// TwinCAT 3 PLC project PLC1
// ProgramVersion: 3.1.4026.24
// libraries:
//   Tc2_MC2, * (Beckhoff Automation GmbH)
//   Tc2_Standard, * (Beckhoff Automation GmbH)
//   Tc2_System, * (Beckhoff Automation GmbH)
//   Tc3_Mc3PlanarMotion, * (Beckhoff Automation GmbH)
//   Tc3_Physics, * (Beckhoff Automation GmbH)
//   Tc3_XPlanarUtility, * (Beckhoff Automation GmbH)
//   XPlanarApplication, * (Beckhoff Automation LLC)
// project tree:
//   GVLs/ GVL.TcGVL (not stored)
//   / PlcTask.TcTTO (not stored)
//   POUs/ MAIN.TcPOU
//   POUs/Utilities/ ErrorStep.TcPOU (not stored), NextMinorStep.TcPOU (not stored), NextStep.TcPOU (not stored)
//   POUs/XPlanarModule/ FB_XPlanarModule.TcPOU
// real-time tasks:
//   TASK XPlanar Task_3: cycle T#250us, priority 1, ADS port 350
//   TASK Job Task: cycle default, priority 2
//   TASK MC-Task (MET): cycle T#2ms, priority 3, ADS port 351
//   TASK MC-Task (MPT): cycle T#10ms, priority 4, ADS port 352
//   TASK PlcTask: cycle T#10ms, priority 20, ADS port 353
// variable links:
//   PLC1/PLC1 Instance <-> XPlanar MC Project/Axes/Mover4220_1
//     PlcTask Inputs/MAIN.XPlanarTable.Movers[1]._Mover.MCTOPLC/ACT <-> McToPlc/ACT
//     PlcTask Inputs/MAIN.XPlanarTable.Movers[1]._Mover.MCTOPLC/COORDMODE <-> McToPlc/COORDMODE
//     PlcTask Inputs/MAIN.XPlanarTable.Movers[1]._Mover.MCTOPLC/SET <-> McToPlc/SET
//     PlcTask Inputs/MAIN.XPlanarTable.Movers[1]._Mover.MCTOPLC/SETONTRACK <-> McToPlc/SETONTRACK
//     PlcTask Inputs/MAIN.XPlanarTable.Movers[1]._Mover.MCTOPLC/STD <-> McToPlc/STD
//     PlcTask Outputs/MAIN.XPlanarTable.Movers[1]._Mover.PLCTOMC/STD <-> PlcToMc/STD
//   PLC1/PLC1 Instance <-> XPlanar MC Project/Groups/Environment
//     PlcTask Inputs/XPlanar.Environment.MCTOPLC_STD <-> McToPlc/STD
//   PLC1/PLC1 Instance <-> XPlanar MC Project/Groups/Track1
//     PlcTask Inputs/MAIN.XPlanarTable.Tracks[1]._Track.MCTOPLC_STD <-> McToPlc/STD
//   PLC1/PLC1 Instance <-> XPlanar MC Project/Groups/Track2
//     PlcTask Inputs/MAIN.XPlanarTable.Tracks[2]._Track.MCTOPLC_STD <-> McToPlc/STD
//   PLC1/PLC1 Instance <-> XPlanar MC Project/Groups/XPlanar
//     PlcTask Inputs/XPlanar.Group.MCTOPLC_STD <-> McToPlc/STD
//   TcCOM Objects/XPlanar/Mover4220_1 <-> XPlanar MC Project/Axes/Mover4220_1
//     InputsFromNC3/NC3ToHW <-> McToIo/STD
//     OutputsToNC3/HWToNC3 <-> IoToMc/STD

// ---- POUs/MAIN.TcPOU
PROGRAM MAIN
VAR
	XPlanarTable : FB_XPlanarModule;
	Initialize	 : BOOL; // Initialize the system
	Reset		 : BOOL; // Reset and Execute System
	Start		 : BOOL; // Run the system
	Halt		 : BOOL; // Avoid Disabling while spinning, otherwise physical sqauring of mover is required
	MachineState : (Startup,
		InitSystem,
		ResetSystem,
		Recover,
		Ready,
		Run,
		Disable);
	trig : R_TRIG;
END_VAR

//This project is an example that shows how you can build track segments using PLC logic
//The specific code for this is in the BuildTracks method of FB_XPlanarModule
//It is a working sample the builds the tracks during the Reset state, joins the mover to the track and runs 1 loop.


//Keep all XPlanar motion system objects up to date every cycle
XPlanarTable.CyclicLogic();


// "Machine" Sequence
CASE MachineState OF
	Startup:	
		IF Initialize THEN
			Initialize := FALSE;
			MachineState := InitSystem;
		END_IF
	
	InitSystem:	
		IF XPlanarTable.Initialize() THEN
			MachineState := ResetSystem;
		END_IF
	
	ResetSystem:	
		IF Reset AND_THEN XPlanarTable.Reset() THEN
			Reset := FALSE;
			MachineState := Recover;
		END_IF
	
	Recover:	
		IF XPlanarTable.Recovery() THEN
			MachineState := Ready;
		END_IF
		
	Ready:
		IF Start THEN
			MachineState := Run;
		END_IF
	
	Run: 
		XPlanarTable.Execute();
	
	Disable:	
		IF XPlanarTable.Disable() THEN
			MachineState := 0;
		END_IF
END_CASE

IF Halt OR trig.Q THEN
	MachineState := Disable;
	Halt := FALSE;
END_IF

END_PROGRAM

// ---- POUs/XPlanarModule/FB_XPlanarModule.TcPOU
FUNCTION_BLOCK FB_XPlanarModule
VAR CONSTANT
	MoverCount	 : UDINT := 1;
	TrackCount	 : UDINT := 2;
END_VAR

VAR
	XPlanarSystem	: FB_Component_XPlanar;
	Movers			: ARRAY[1..MoverCount] OF FB_XPlanarMover;
	Tracks			: ARRAY[1..TrackCount] OF FB_XPlanarTrackSegment;
	InitState		: (CheckForXPlanarInit, UpdateDynamics, SetStationParameters, Initialized);
END_VAR

METHOD BuildTracks : BOOL

VAR_INST
	TrackIndex	: UDINT;
	TaskResult	: I_PlanarTaskResult;
END_VAR

VAR
	i : UDINT;
	AllTracksCleared	: BOOL;
END_VAR
CASE TrackIndex OF
	0:
		//Clear any old track data
		AllTracksCleared := TRUE;
		FOR i := 1 TO TrackCount DO
			TaskResult := Tracks[i].Clear();
			IF NOT TaskResult.Done THEN
				AllTracksCleared := FALSE;
			END_IF
		END_FOR

		IF AllTracksCleared THEN
			TrackIndex := 1;
		END_IF

// *You can add up to 20 geometric items by default.  If more are required you can increase the value in SystemParameters
	1: //Add geometric points for track 1.  
		//
		Tracks[TrackIndex].Definition.Items[1].ItemType := XPlanarApplication.E_TrackItemType.Line;
		Tracks[TrackIndex].Definition.Items[1].StartPoint.SetValuesXY(180, 320);
		Tracks[TrackIndex].Definition.Items[1].EndPoint.SetValuesXY(180, 100);

		//
		Tracks[TrackIndex].Definition.Items[2].ItemType := XPlanarApplication.E_TrackItemType.Line;
		Tracks[TrackIndex].Definition.Items[2].StartPoint.SetValuesXY(140, 60);
		Tracks[TrackIndex].Definition.Items[2].EndPoint.SetValuesXY(100, 60);

		//Build the track segment with the configured points
		TaskResult := Tracks[TrackIndex].Build();
		
		//If Successful move on to the next segment
		IF TaskResult.Done THEN
			IF TrackIndex < TrackCount THEN
				TrackIndex := TrackIndex + 1;
			ELSE
				TrackIndex	:= 0;	 //Reset the Index var
				BuildTracks := TRUE; //Return TRUE that all tracks were built successfully
			END_IF
		END_IF

	2: //Add geometric points for track 2
		//
		Tracks[TrackIndex].Definition.Items[1].ItemType := XPlanarApplication.E_TrackItemType.Line;
		Tracks[TrackIndex].Definition.Items[1].StartPoint.SetValuesXY(60, 100);
		Tracks[TrackIndex].Definition.Items[1].EndPoint.SetValuesXY(60, 320);

		//
		Tracks[TrackIndex].Definition.Items[2].ItemType := XPlanarApplication.E_TrackItemType.Line;
		Tracks[TrackIndex].Definition.Items[2].StartPoint.SetValuesXY(100, 360);
		Tracks[TrackIndex].Definition.Items[2].EndPoint.SetValuesXY(140, 360);

		//Set any connecting tracks for this segment.  Segments must already be built!
		Tracks[TrackIndex].Definition.StartFromTrackID := 1;
		Tracks[TrackIndex].Definition.EndAtTrackID	   := 1;

		//Build the track segment with the configured points
		TaskResult := Tracks[TrackIndex].Build();
		
		//If Successful move on to the next segment
		IF TaskResult.Done THEN
			IF TrackIndex < TrackCount THEN
				TrackIndex := TrackIndex + 1;
			ELSE
				TrackIndex	:= 0;	 //Reset the Index var
				BuildTracks := TRUE; //Return TRUE that all tracks were built successfully
			END_IF
		END_IF
END_CASE
END_METHOD

METHOD CyclicLogic : BOOL
VAR
	i : UDINT;
END_VAR
VAR_INST
	TaskResult	: I_PlanarTaskResult;
END_VAR
XPlanarSystem.CyclicLogic();
IF NOT XPlanarSystem.Initialized THEN
	RETURN;
END_IF

//Add any logic that needs to be called every cycle here
END_METHOD

METHOD Disable : BOOL
VAR_INST
	CommandResult	: I_PlanarTaskResult;
END_VAR
CommandResult := XPlanarSystem.Abort(); // Stop Motion and Disable All Movers
IF CommandResult.Done THEN
	Disable := TRUE;
END_IF
END_METHOD

METHOD Execute : BOOL
VAR
	i : UDINT;
END_VAR

VAR_INST
	runloop: BOOL := TRUE;
END_VAR
//The XPlanar system is now 'running' put necessary run logic here

IF runloop THEN
	Movers[1].MoveCommand.TrackMoveXY(120, 60, 150, Tracks[1], XPlanarApplication.MC_DIRECTION.mcDirectionPositive);
	runloop := FALSE;
END_IF
END_METHOD

METHOD Initialize : BOOL
VAR_INST
	i			: UDINT;
END_VAR
CASE InitState OF
	CheckForXPlanarInit: // Init Vars
		Initialize := FALSE;
		
		//Make sure the XPlanar motion system has initialized
		IF XPlanarSystem.Initialized THEN
			InitState := UpdateDynamics;
		END_IF

	UpdateDynamics: 
		//Assign Initial Application Mover Dynamics
		FOR i := 1 TO XPlanar.MoverCount DO
			ip.Movers[i].Gap						:= 200;
			ip.Movers[i].Dynamics.Movement.Velocity := GVL.MoverVelo;
			ip.Movers[i].Dynamics.Movement.Accel	:= GVL.MoverVelo * 10;
			ip.Movers[i].Dynamics.Movement.Decel	:= GVL.MoverVelo * 10;
			ip.Movers[i].Dynamics.Movement.Jerk		:= GVL.MoverVelo * 100;
			ip.Movers[i].Dynamics.Rotation.Velocity := GVL.MoverSpinVelo;
			ip.Movers[i].Dynamics.Rotation.Accel	:= GVL.MoverSpinVelo * 10;
			ip.Movers[i].Dynamics.Rotation.Decel	:= GVL.MoverSpinVelo * 10;
			ip.Movers[i].Dynamics.Rotation.Jerk		:= GVL.MoverSpinVelo * 100;
		END_FOR

		InitState := Initialized;

	Initialized: // Init Complete
		Initialize := TRUE;
END_CASE
END_METHOD

METHOD Recovery : BOOL
VAR_INST
	RecoverState	: UDINT;
	ipResult		: ARRAY[1..MoverCount] OF I_PlanarTaskResult;
	ErrorMoverId, i : UDINT;
	ItemsOk			: BOOL;
END_VAR
//This is an example of some very simple mover recovery.  
//What needs to be done to recover will be unique for each application.

CASE RecoverState OF
	0: // Init Vars
		Recovery := FALSE;
		i := 1;
		NextStep(RecoverState);
		
	10: // All Movers Join rack closest to their current location
		IF i <= XPlanar.MoverCount THEN
			ipResult[i] := ip.Movers[i].MoveCommand.JoinClosestTrack(FALSE);
			IF ipResult[i].Done THEN
				NextMinorStep(RecoverState);
			ELSIF ipResult[i].Error THEN
				ErrorStep(RecoverState);
			END_IF
		ELSE
			i := 1;
			NextStep(RecoverState);
		END_IF

	11: //Check Mover Count
		IF i <= XPlanar.MoverCount THEN
			i	   := i + 1;
			RecoverState := 10;
		ELSE
			i := 1;
			NextStep(RecoverState);
		END_IF

	20: // Complete
		RecoverState		 := 0;
		ErrorMoverId := 0;
		Recovery	 := TRUE;
END_CASE
END_METHOD

METHOD Reset : BOOL
VAR_INST
	ResetState	  : UDINT;
	i			  : UDINT;
	ResetOk		  : BOOL;
	ResetError	  : BOOL;
	CommandResult : I_PlanarTaskResult;
END_VAR
CASE ResetState OF
	0: // Init Vars
		Reset := FALSE;
		NextStep(ResetState);

	10: // Reset Table 
		IF XPlanarSystem.Reset().Done THEN
			NextStep(ResetState);
		END_IF
		
	20: //Build Track Segments
		IF BuildTracks() THEN
			NextStep(ResetState);
		END_IF

	30: // Enable Movers
		CommandResult := XPlanarSystem.EnableMovers();
		IF CommandResult.Done THEN
			NextStep(ResetState);
		ELSIF CommandResult.Error THEN
			ErrorStep(ResetState);
		END_IF

	40: // Add Movers To Group
		CommandResult := XPlanarSystem.AddMoversToGroup();
		IF CommandResult.Done THEN
			NextStep(ResetState);
		ELSIF CommandResult.Error THEN
			ErrorStep(ResetState);
		END_IF

	50: // Enable Tracks
		CommandResult := XPlanarSystem.EnableTracks();
		IF CommandResult.Done THEN
			NextStep(ResetState);
		ELSIF CommandResult.Error THEN
			ErrorStep(ResetState);
		END_IF

	60: // Add Tracks To Group
		CommandResult := XPlanarSystem.AddTracksToGroup();
		IF CommandResult.Done THEN
			NextStep(ResetState);
		ELSIF CommandResult.Error THEN
			ErrorStep(ResetState);
		END_IF

	70: // Enable Group
		CommandResult := XPlanarSystem.EnableGroup();
		IF CommandResult.Done THEN
			NextStep(ResetState);
		ELSIF CommandResult.Error THEN
			ErrorStep(ResetState);
		END_IF

	80: // Complete
		Reset  := TRUE;
		ResetState := 0;
END_CASE
END_METHOD

END_FUNCTION_BLOCK
